# EPICS alarm handler configuration: mps_database/bareTest/alarms/areas/mpln_sph_mp01.alhConfig
GROUP NULL MPLN:SPH:MP01:1
$ALIAS MPS Link Node 120
$GUIDANCE
LTUH MPS
   Group Name: MPLN:SPH:MP01:1
   Summary PV:  MPLN:SPH:MP01:1:STATSUMY
$END
CHANNEL  MPLN:SPH:MP01:1    MPLN:SPH:MP01:1:MPS_EN_RBV		-----
CHANNEL  MPLN:SPH:MP01:1    MPLN:SPH:MP01:1:LC1_MODE_RBV		-----
